TYPE ST_MKS_909 EXTENDS ST_VacuumGauge:
STRUCT

	//Discrete Control: Ion gauges only
	i_xHvOn	:	BOOL;//High voltage On to turn on this Hot Cathode gauge, they turn on immediately, unlike cold cathodes
	
END_STRUCT
END_TYPE

(* stored: Version 1.1.0.1, ProductVersion 3.1.4020.12
   DUT ST_MKS_909: Id {2d5baa0e-8e32-47a1-a5af-5d0c881a9361} *)
